{attribute 'qualified_only'}
VAR_GLOBAL
(* Buffer Variable *)
RxBufferPcCom		: ComBuffer;	(* Receive data buffer; used with all receive function blocks *)
TxBufferPcCom		: ComBuffer;	(* Transmit data buffer; used with all receive function blocks *)
END_VAR

(* stored: Version 1.1.0.1, ProductVersion 3.1.4024.11
   GVL SerialComm: Id {79362f68-9ccc-4fc0-beb6-ddf610e22780} *)
